ABB RAPID module: HSLU_Workobject.modx

MODULE HSLU_Workobject

    !***********************************************************************************
    !
    ! Digital Construction
    ! Hochschule Luzern - Technik & Architektur
    ! Technikumstrasse 21
    ! CH-6048 Horw
    !
    !***********************************************************************************
    !
    ! PROJECT     :  Swissbau
    !
    ! FUNCTION    :  Workobject
    !
    ! AUTHOR      :  Juri Jerg
    !
    ! EMAIL       :  juri.jerg@hslu.ch
    !
    ! HISTORY     :  2025.12.28
    !
    ! Copyright   :  HSLU (2025)
    !
    !***********************************************************************************

    !************************************************
    ! Declaration :     wobjdata
    !************************************************
    !

    TASK PERS wobjdata ob_HSLU_Pick_small_old := [FALSE,TRUE,"",[[447.9645,-686.7764,-35.14248],[0.705938,0.001679464,-0.002182502,-0.7082683]],[[0,0,0],[1,0,0,0]]]; !EAX 1000mm
    TASK PERS wobjdata ob_HSLU_Pick_medium_old := [FALSE,TRUE,"",[[447.9645,-386.7764,-35.14248],[0.705938,0.001679464,-0.002182502,-0.7082683]],[[0,0,0],[1,0,0,0]]]; !EAX 700mm
    TASK PERS wobjdata ob_HSLU_Pick_large_old := [FALSE,TRUE,"",[[447.9645,313.2236,-35.14248],[0.705938,0.001679464,-0.002182502,-0.7082683]],[[0,0,0],[1,0,0,0]]]; !EAX 0mm
    TASK PERS wobjdata ob_HSLU_Cut_old := [FALSE,TRUE,"",[[449.3956,-1103.482,-34.07918],[0.707108856,0.002987127,-0.006913478,-0.707064599]],[[15,230,72.161],[1,0,0,0]]]; !EAX 500mm
    TASK PERS wobjdata ob_HSLU_Place_old := [FALSE,TRUE,"",[[492,0,2],[0.708136408,-0.000931269,-0.001221202,0.706073983]],[[0,0,-1],[1,0,0,0]]];
    TASK PERS wobjdata ob_HSLU_Glue_old := [FALSE,TRUE,"",[[332.557,-885.513,1275.448],[0,0.707106781,0.707106781,0]],[[-14.734,13.382,12.742],[1,0,0,0]]]; !EAX 200mm
    TASK PERS wobjdata ob_HSLU_Lable_old := [FALSE,TRUE,"",[[369.499,-1204.703,942.427],[0.003085325,-0.70710005,-0.70710005,0.003085325]],[[-40.132,11.963,3.574],[1,0,0,0]]]; !EAX 350mm


    TASK PERS wobjdata ob_HSLU_Pick_small := [FALSE,TRUE,"",[[446.6452,-691.3218,-39.81755],[0.7071373,-0.0003829703,0.001478308,-0.7070746]],[[0,0,0],[1,0,0,0]]]; !EAX 1000mm
    TASK PERS wobjdata ob_HSLU_Pick_medium := [FALSE,TRUE,"",[[446.6452,-391.3218,-39.81755],[0.7071373,-0.0003829703,0.001478308,-0.7070746]],[[0,0,0],[1,0,0,0]]]; !EAX 700mm
    TASK PERS wobjdata ob_HSLU_Pick_large := [FALSE,TRUE,"",[[446.6452,308.6782,-39.81755],[0.7071373,-0.0003829703,0.001478308,-0.7070746]],[[0,0,0],[1,0,0,0]]]; !EAX 0mm
    TASK PERS wobjdata ob_HSLU_Cut_Top := [FALSE,TRUE,"",[[452.1468,-1099.857,-41.04398],[0.7080513,-0.000488674,-0.001296379,-0.7061597]],[[17.50001382,230.003717517,102.161],[0.99999309,0,0,-0.003717543]]]; !EAX 500mm
    TASK PERS wobjdata ob_HSLU_Cut_Back := [FALSE,TRUE,"",[[452.1468,-1099.857,-41.04398],[0.7080513,-0.000488674,-0.001296379,-0.7061597]],[[17.50001382,100,18],[0.99999309,0,0,-0.003717543]]]; !EAX 500mm
    !TASK PERS wobjdata ob_HSLU_Place := [FALSE,TRUE,"",[[492,0,-3],[0.707103595,0.002122708,0.002122708,0.707103595]],[[0,0,-1],[1,0,0,0]]];
    TASK PERS wobjdata ob_HSLU_Place := [FALSE,TRUE,"",[[492,0,-3],[0.707095615,0.003973891,0.003973891,0.707095615]],[[0,0,-1],[1,0,0,0]]];
    TASK PERS wobjdata ob_HSLU_Glue := [FALSE,TRUE,"",[[343.930,-1182.871,1270.578],[0,0.707106781,0.707106781,0]],[[-14.734,13.382,22.742],[1,0,0,0]]]; !EAX 500mm
    TASK PERS wobjdata ob_HSLU_Lable := [FALSE,TRUE,"",[[376.691,-1205.025,934.740],[0.003085325,-0.70710005,-0.70710005,0.003085325]],[[-40.132,11.963,3.574],[1,0,0,0]]]; !EAX 350mm

    TASK PERS wobjdata ob_HSLU_Pick_400 := [FALSE,TRUE,"",[[446.6452,58.6782,-35.14248],[0.705938,0.001679464,-0.002182502,-0.7082683]],[[0,0,0],[1,0,0,0]]]; !EAX 250mm
    TASK PERS wobjdata ob_HSLU_Pick_550 := [FALSE,TRUE,"",[[446.6452,-591.3218,-35.14248],[0.705938,0.001679464,-0.002182502,-0.7082683]],[[0,0,0],[1,0,0,0]]]; !EAX 900mm
    TASK PERS wobjdata ob_HSLU_Pick_750 := [FALSE,TRUE,"",[[446.6452,-491.3218,-35.14248],[0.705938,0.001679464,-0.002182502,-0.7082683]],[[0,0,0],[1,0,0,0]]]; !EAX 800mm
    TASK PERS wobjdata ob_HSLU_Pick_1000 := [FALSE,TRUE,"",[[446.6452,308.6782,-35.14248],[0.705938,0.001679464,-0.002182502,-0.7082683]],[[0,0,0],[1,0,0,0]]]; !EAX 0mm

ENDMODULE
